// TIA Portal V21 export
VAR_GLOBAL   // PLC tag table "K_Num"
END_VAR
VAR_GLOBAL CONSTANT   // user constants
   K_NumAnalogica : Int := 0;
   K_NumComunicazione : Int := 0;
   K_NumComunicazioneS7 : Int := 0;
   K_NumConsenso : Int := 0;
   K_NumDispositivoProfinet : Int := 0;
   K_NumMacchinaARicetta : Int := 0;
   K_NumMotore : Int := 0;
   K_NumParatia : Int := 0;
   K_NumPid : Int := 0;
   K_NumPortata : Int := 0;
   K_NumSegnaliMacchina : Int := 0;
   K_NumSensore : Int := 0;
   K_NumSequenza : Int := 0;
   K_NumValvola : Int := 0;
END_VAR
